FUNCTION_BLOCK FB_PowerQualityMonitoring
VAR PERSISTENT
	r_BESSEnergySupplied		: REAL;
	r_BESSEnergyConsumed		: REAL;
END_VAR


VAR_OUTPUT
	get							: ST_PowerMonitor_get;
END_VAR

VAR_INPUT
	b_Enable					: 	BOOL;
	PowerStackGet				:	st_Powerstack_Get;
	b_TNModeActive				:	BOOL;
	b_ThirdOutputFieldAvailable	: 	BOOL;
	b_InputFieldsAvailable		: 	BOOL;
	b_NeutralTransformerAvailable: BOOL;
END_VAR

VAR
	Janitza	: FB_Janitza;
	El3443	: FB_EL34xx := (VoltageRatio := 1, CurrentRatio := 1);
END_VAR

(*
Update rate is 200 ms max.
So call IO method only every 200ms.
More calls only increase cpu and network load.
*)

//get data from janitza powermeter
Janitza(
	get:=get, 
	ReadData:=b_Enable, 
	b_TNmodeEnable := b_TNModeActive,
	b_NeutralTransformerAvailable := b_NeutralTransformerAvailable,
	b_ThirdOutputFieldAvailable := b_ThirdOutputFieldAvailable,
	b_InputFieldsAvailable := b_InputFieldsAvailable,
	);
EL3443();

MapPowerstackGetToGetStruct();

MapEL3443OutputToGetStruct();

//MapCEEOutputToGetStruct(); // FIX NAN --> RUNTIME EXEPTION!!!

CalcBessEnergyValues();

GetLoadshares(powerstackGet.r_RatedPower, get.InputField.ar_ApparentPower[0], get.OutputField.ar_ApparentPower[0]);

METHOD CalcBessEnergyValues : BOOL

VAR_INST
	ton_CumEnergy		: TON := (PT:= T#100ms);
END_VAR
ton_CumEnergy(IN:= NOT ton_CumEnergy.Q);

IF ton_CumEnergy.Q THEN
	IF get.BESS.r_ActivePower > 0 THEN
		r_BESSEnergySupplied := r_BESSEnergySupplied + ABS(get.BESS.r_ActivePower) / 36000;
	ELSIF get.BESS.r_ActivePower < 0 THEN
		r_BESSEnergyConsumed := r_BESSEnergyConsumed + ABS(get.BESS.r_ActivePower) / 36000;
	END_IF	
END_IF


//Set persistent values to get struct.
Get.BESS.r_EnergySupplied := r_BESSEnergySupplied;
Get.BESS.r_EnergyConsumed := r_BESSEnergyConsumed;
END_METHOD

METHOD PUBLIC EMstop : BOOL
//returns true when ready/stopped
END_METHOD

METHOD EnergyBalance : REAL
VAR_INPUT
	IN1	: REAL;
	IN2 : REAL;
	IN3 : REAL;
END_VAR
EnergyBalance := IN1 + IN2 + IN3;
END_METHOD

METHOD GetDiagnostics
VAR_IN_OUT
	AddError		: ARRAY [*] OF FB_AddErrorST;
	a_ActiveEvents	: ARRAY [*] OF ST_ErrorStruct;
	w_Index			: WORD;
END_VAR
//JANITZA
(*Comm Warning*)		AddError[w_Index](
		b_ErrorTrig			:= get.events.b_MBCommWarning,
		out_ST_Error			:= a_ActiveEvents[w_Index],
		w_ErrorID					:= 1,
		e_ObjectID				:= eObject_ID.PowerMonitor,
		s_Message				:= 'janitza communication warning',
		e_sev					:= eseverity.warning
	);
	w_Index := w_Index +1;
	
(*Comm timeout*)		AddError[w_Index](
		b_ErrorTrig			:= get.events.b_MBTimeoutWarning,
		out_ST_Error			:= a_ActiveEvents[w_Index],
		w_ErrorID					:= 2,
		s_Message				:= 'janitza communication timeout',
		e_sev					:= eseverity.Warning
	);
	w_Index := w_Index +1;
	
(*Comm fault*)		AddError[w_Index](
		b_ErrorTrig			:= get.events.b_MBCommError,
		out_ST_Error			:= a_ActiveEvents[w_Index],
		w_ErrorID					:= 3,
		t_TriggerTime		:= T#10S,
		s_Message				:= 'janitza communication fault',
		e_sev					:= eseverity.Normalshutdown
	);
	w_Index := w_Index +1;
	
//EL3443
(*Comm Warning*)		AddError[w_Index](
		b_ErrorTrig			:= get.events.b_EL3443Warning,
		out_ST_Error			:= a_ActiveEvents[w_Index],
		w_ErrorID					:= 4,
		s_Message				:= 'EL3443 powermonitor warning',
		e_sev					:= eseverity.Warning,
	);
	w_Index := w_Index +1;
END_METHOD

METHOD GetLoadshares : BOOL
VAR_INPUT
	r_ratedPower		: REAL;
	r_InputPower		: REAL;
	r_OutputPower		: REAL;
END_VAR
get.InputField.r_loadshare := r_InputPower / MAX(1, r_ratedPower) * 100;
get.OutputField.r_loadshare := r_OutputPower /  MAX(1, r_ratedPower) * 100;
END_METHOD

METHOD MapCEEOutputToGetStruct : BOOL
VAR_INPUT
END_VAR
VAR_INST
	r_CEEPower : REAL;
END_VAR
//r_CEEPower := - Get.InputField.ar_ActivePower[0] - Get.OutputField.ar_ActivePower[0] + Get.BESS.r_ActivePower;
//Get.CEE.r_ReactivePower := - Get.InputField.r_ReactivePhasePower[0] - Get.OutputField.r_ReactivePhasePower[0] + Get.BESS.r_ReactivePower;
//Get.CEE.r_ApparentPower := SQRT(EXPT(Get.CEE.r_ActivePower, 2) + EXPT(Get.CEE.r_ReactivePower,2));
//Get.CEE.r_Current[0] := SEL(Get.OutputField.r_LineVoltage[0] = 0, Get.CEE.r_ApparentPower * 1000 / MAX(1, Get.OutputField.r_LineVoltage[0] * 1.73), 0); 
//Get.CEE.r_PowerFactor := LIMIT(-1, ABS(Get.CEE.r_ApparentPower / MAX(1,Get.CEE.r_ActivePower)) * SEL(Get.CEE.r_ReactivePower <0, -1,1), 1);
END_METHOD

METHOD MapEL3443OutputToGetStruct
IF b_Enable THEN
	IF EL3443.ui_EL3443BoxState = 16#8 THEN //EL3443.TotalStatus.bit_SystemState AND 
		//Get Generator field voltage data from EL3443
		Get.InputField.ar_PhaseVoltage[Phases.L1]:= EL3443.r_PhaseVoltage[Phases.L1];
		Get.InputField.ar_PhaseVoltage[Phases.L2]:=  EL3443.r_PhaseVoltage[Phases.L2];
		Get.InputField.ar_PhaseVoltage[Phases.L3]:=  EL3443.r_PhaseVoltage[Phases.L3];
		Get.InputField.ar_PhaseVoltage[Phases.AVG] := EL3443.r_PhaseVoltage[0];
		get.InputField.li_TimeVoltZeroCrossup := EL3443.li_TimeVoltZeroCrossup;
		
		Get.InputField.ar_LineVoltage[Phases.L1]:=  EL3443.r_LineVoltage[Phases.L1];
		Get.InputField.ar_LineVoltage[Phases.L2]:=  EL3443.r_LineVoltage[Phases.L2];
		Get.InputField.ar_LineVoltage[Phases.L3]:=  EL3443.r_LineVoltage[Phases.L3];
		Get.InputField.ar_LineVoltage[Phases.AVG] := EL3443.r_LineVoltage[0];
		
		Get.InputField.ar_Frequency[0] :=  EL3443.r_Frequency;
		
		Get.InputField.ar_Current[Phases.L1]:= EL3443.r_Current[Phases.L1];
		Get.InputField.ar_Current[Phases.L2]:= EL3443.r_Current[Phases.L2];
		Get.InputField.ar_Current[Phases.L3]:= EL3443.r_Current[Phases.L3];
		Get.InputField.ar_Current[Phases.AVG]:= EL3443.r_Current[Phases.AVG];
		Get.InputField.ar_Current[Phases.N]:= EL3443.r_Current[Phases.N];
		
		Get.InputField.ar_ActivePower[Phases.L1]:= EL3443.r_ActivePower[Phases.L1];
		Get.InputField.ar_ActivePower[Phases.L2]:= EL3443.r_ActivePower[Phases.L2];
		Get.InputField.ar_ActivePower[Phases.L3]:= EL3443.r_ActivePower[Phases.L3];
		Get.InputField.ar_ActivePower[0]:= EL3443.r_ActivePower[0];		
		
		Get.InputField.ar_ApparentPower[Phases.L1]:= EL3443.r_ApparentPower[Phases.L1];
		Get.InputField.ar_ApparentPower[Phases.L2]:= EL3443.r_ApparentPower[Phases.L2];
		Get.InputField.ar_ApparentPower[Phases.L3]:= EL3443.r_ApparentPower[Phases.L3];	
		Get.InputField.ar_ApparentPower[0]	:= EL3443.r_ApparentPower[0];		
		
		// TEMPORARY FIX: 
		Get.InputField.ar_ReactivePower[Phases.L1]:= EL3443.r_ReactivePower[Phases.L1];
		Get.InputField.ar_ReactivePower[Phases.L2]:= EL3443.r_ReactivePower[Phases.L2];
		Get.InputField.ar_ReactivePower[Phases.L3]:= EL3443.r_ReactivePower[Phases.L3];		
		Get.InputField.ar_ReactivePower[Phases.AVG]:= EL3443.r_ReactivePower[0];
		
		//Powerfactors                                                                 
	    Get.InputField.ar_PowerFactor[Phases.L1]:= EL3443.r_PowerFactor[Phases.L1];
		Get.InputField.ar_PowerFactor[Phases.L2]:= EL3443.r_PowerFactor[Phases.L2];
		Get.InputField.ar_PowerFactor[Phases.L3]:= EL3443.r_PowerFactor[Phases.L3];		
		Get.InputField.ar_PowerFactor[Phases.AVG]:= Get.InputField.ar_ActivePower[0] / MAX(1, ABS(Get.InputField.ar_ApparentPower[0])) * SEL(Get.InputField.ar_ReactivePower[0] > 0, 1, -1);             

		//THD not in EL3443                                                       
		get.InputField.r_VoltageUnbalance := EL3443.r_VoltageUnbalance;
		
		//EL3443 only gives a boolean for fieldRotation with True meaning right.
		//So false could be none or left. Check voltages before checking rotation.
		IF (Get.InputField.ar_LineVoltage[Phases.L1] > 300) AND (Get.InputField.ar_LineVoltage[Phases.L2] > 300) AND (Get.InputField.ar_LineVoltage[Phases.L3] > 300) THEN
			IF EL3443.TotalStatus.bit_GridDirection THEN
				Get.InputField.e_ACrotationStatus := eACRotationState.Right;
			ELSE
				Get.InputField.e_ACrotationStatus := eACRotationState.Left;	
			END_IF
		ELSE
			Get.InputField.e_ACrotationStatus := eACRotationState.None;	
		END_IF
		get.events.b_EL3443Warning := FALSE;	
	END_IF
	
	ELSE
		//faultwarning sets directly if the card states an error.
		//Fault error only sets if the fault remains for a longer period of time.
		get.events.b_EL3443Warning := TRUE;
END_IF
END_METHOD

METHOD MapPowerstackGetToGetStruct
//Voltage dependent values of Internal supply are copied from outputfield, but are only valid if netcontactor is closed.
IF powerstackget.Netcontactor.b_NetConFb THEN
	get.BESS.r_LineVoltage := powerstackGet.r_ACVoltageD7;
	get.BESS.r_Frequency := powerstackGet.r_FrequencyD7;
	get.OutputField.ar_Frequency[0] := powerstackGet.r_FrequencyD7;
ELSE
	get.BESS.r_LineVoltage := powerstackGet.r_ACVoltageSupply;
	get.BESS.r_Frequency := powerstackGet.r_FrequencySupply;
END_IF

//Fill BESS data with PowerStackData
//Not all data is filled in here, determine which are desired and possible.
get.BESS.e_ACrotationStatus := get.OutputField.e_ACrotationStatus;
//phase currents not available at this time, only the average is set
get.BESS.ar_Current[0] := PowerStackGet.r_AcCurrent;

//phase Powers not available at this time, only the average is set
Get.BESS.r_ApparentPower	:=	PowerStackGet.r_ApparentPower;
Get.BESS.r_ReactivePower	:=	PowerStackGet.r_ReactivePower;
Get.BESS.r_ActivePower		:=	PowerStackGet.r_ActivePower;


//phase Powerfactors not available at this time, only the average is set									
Get.BESS.r_PowerFactor		:=	PowerStackGet.r_CosPhi;
END_METHOD

METHOD Public Reset : BOOL
//clear data struct
//reinitialize janitza + el3443
//clear all errors?

//returns true when ready
Reset := NOT get.events.b_MBCommError;
END_METHOD

END_FUNCTION_BLOCK

(* stored: Version 1.1.0.1, ProductVersion 3.1.4024.12
   POU FB_PowerQualityMonitoring: Id {e1af34d5-6ad2-44c9-b24a-c806b8db8e6d}, SpecialFunc None
   Method CalcBessEnergyValues: Id {8fffab80-6a89-4a59-b1b7-39f5740c568f}
   Method EMstop: Id {02287e66-26ae-4c64-a18d-2c9f331ba2dd}
   Method EnergyBalance: Id {814f7b21-138c-419b-ad9b-671fe21399c2}
   Method GetDiagnostics: Id {3affa096-4b6f-49ac-a980-75c93b2f7449}
   Method GetLoadshares: Id {53760293-9558-413f-839b-df58c21753a1}
   Method MapCEEOutputToGetStruct: Id {3ac2b540-d8a9-436a-a149-02a7b22497d0}
   Method MapEL3443OutputToGetStruct: Id {b858e6d2-878c-401f-bd99-882eaa16aed5}
   Method MapPowerstackGetToGetStruct: Id {220670fd-2d02-40a2-8be2-89d58383bcf5}
   Method Reset: Id {f0888ded-5a81-4f63-8a49-a3d35f7817a5} *)
